PROGRAM SHA1_MD5_DEMO_1
VAR
	text: STRING(STRING_LENGTH) := '<4036.1076324381@guildenstern.zeitform.de>';
	MD5_STR : MD5_STR;
	SHA1_STR : SHA1_STR;
	md5_hash : ARRAY [0..15] OF BYTE;
	sha1_hash : ARRAY [0..19] OF BYTE;
	start1 : BOOL := TRUE;
	start2 : BOOL := TRUE;
	done1 : BOOL;
	done2 : BOOL;
	md5_strh : STRING(32);
	sha1_strh : STRING(40);
END_VAR

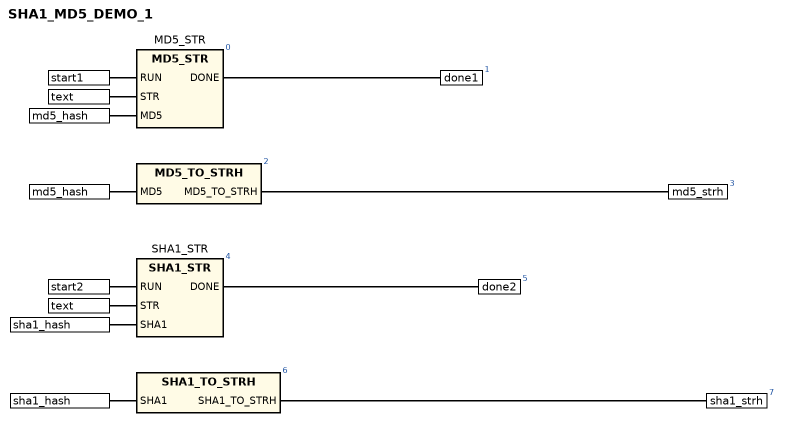
MD5_STR(RUN := start1, STR := text, MD5 := md5_hash);
done1 := MD5_STR.DONE;
md5_strh := MD5_TO_STRH(MD5 := md5_hash);
SHA1_STR(RUN := start2, STR := text, SHA1 := sha1_hash);
done2 := SHA1_STR.DONE;
sha1_strh := SHA1_TO_STRH(SHA1 := sha1_hash);

END_PROGRAM

(* stored: Version 1.1.0.1, ProductVersion 3.1.4024.0
   POU SHA1_MD5_DEMO_1: Id {fb465035-cf2e-4437-9a0f-88663a74c536}, SpecialFunc None *)
